# EPICS substitutions: tpmacApp/Db/autohome.substitutions
file "db/autohome.db"
{
pattern
{SYS,            DEV,                  PLC,  PORT  }
{"XF:03IDC-OP",  "{Det:Vort-Ax:X}",    8,    P0    }
{"XF:03IDC-OP",  "{Det:Vort-Ax:Y}",    9,    P0    }
{"XF:03IDC-OP",  "{Det:Vort-Ax:Z}",    10,   P0    }
{"XF:03IDC-OP",  "{Det:Bruk-Ax:X}",    11,   P0    }
{"XF:03IDC-OP",  "{Det:Bruk-Ax:Y}",    12,   P0    }
{"XF:03IDC-OP",  "{Det:Bruk-Ax:Z}",    13,   P0    }
{"XF:03IDC-OP",  "{Det:Bruk-Ax:7}",    14,   P0    }
{"XF:03IDC-OP",  "{Det:Bruk-Ax:8}",    15,   P0    }
}
